Fanuc KAREL source: KT00282.KL

PROGRAM KT00282
%NOLOCKGROUP
VAR
  P1: XYZWPR
  P2: JOINTPOS
  OUT: BOOLEAN
BEGIN
  P1.X = 1.0
  OUT = P1 = P2
END KT00282
